Staubli VAL3: cycle_run.pgx

program cycle_run(progItem& x_pProgram[] (dimensions=1))
  local num i
  local num j
  local num l_nClock
  local num l_nResult
  local num l_nSize
  local progItem l_pProg
  local string l_sEvent
begin
  //
  // START
  //
  cycleStatus:nEvent=0
  cycleStatus:nPoint=0
  // refresh
  cycleStatus:pCycleProg=l_pProg=x_pProgram
  // check the cycle
  if cycleStatus:bCycle
    // print the actual program
    call cycleStatus:printLog("[PROG "+l_pProg.sID+"]")
  endIf
  l_nSize=size(l_pProg.iEvent)
  for i=0 to l_nSize-1
    // wait pause false before doing the next instruction
    wait(cycleStatus:bPause==false and isPowered() and cycleStatus:nWorkingStatus==0)
    if l_pProg.iEvent[i].sType!=""
      l_sEvent=l_pProg.iEvent[i].sType+" "+l_pProg.iEvent[i].sData
      if saveData:bDebug
        ? "ACTION READ,"+l_sEvent+",ID="+toString(".3",getMoveId())+","+toString(".3",clock()-cycleStatus:nTime)
      endIf
      call cycle_doEvent(l_pProg.iEvent[i],i)
      // JUMP CALL USED
      call cycle_isCallUse()
      // GOTO USED
      if cycleStatus:bGOTO
        // terminate this and run the GOTO
        i=l_nSize-1
      endIf
    endIf
  endFor
  // GOTO ...
  if cycleStatus:bGOTO
    // INIT
    cycleStatus:bGOTO=false
    call action_wait()
    if cycleStatus:iToSuperV.sType=="PROG"
      // run the GOTO FOR PROG
      call prog:getProgItem(l_pProg,cycleStatus:iToSuperV.sData)
      //use:bUseRefresh=true
      call cycle_run(l_pProg)
    else
      call cycle_doEvent(cycleStatus:iToSuperV,0)
      // JUMP CALL USED
      call cycle_isCallUse()
    endIf
  endIf
end
